# B&R Automation Studio project ControlObjectModeling
Automation Studio 4.2.10.53 SP

## Configuration Config1

CPU 4PP065.0351-P74, AutomationRuntime D4.26, Build 4.1.2, Vc V4.26.5, Safety 0.0

### Task classes (Cpu.sw)
```
Cyclic#2 (cycle 20000 us, tolerance 20000 us):
  Program <- Program.prg
Binaries: TCData, iomap, Role, sysconf, arconfig, asfw, User, ashwd
Libraries: MotorContr
```

### Hardware
```
4PP065_0351_P74 : 4PP065.0351-P74 v1.0.3.0
  Connector IF4:
    EplInterfaceRedundant = 0
    EplEthInterfaceRedundant = 0
  Connector IF5:
    ActivateDevice = 1
  ConfigurationID = Lab1_Config1
  Simulation = 1
  Cyclic1Duration = 10000
  Cyclic1Tolerance = 10000
  Cyclic2Duration = 20000
  Cyclic2Tolerance = 20000
  Cyclic3Duration = 50000
  Cyclic3Tolerance = 50000
  Cyclic4Duration = 100000
  Cyclic4Tolerance = 100000
  Cyclic5Duration = 200000
  Cyclic5Tolerance = 200000
  Cyclic6Duration = 500000
  Cyclic6Tolerance = 500000
  Cyclic7Duration = 1000000
  Cyclic7Tolerance = 1000000
  Cyclic8Duration = 10000
  Cyclic8Tolerance = 30000000
```

## Logical view

Binary libraries used (declarations not repeated): operator, runtime, astime, AsIecCon

### Package Logical/Libraries - Global libraries

### Library Logical/Libraries/MotorContr (ANSIC)

#### MotorContr.fun - Exported functions and function blocks
```iecst
FUNCTION_BLOCK FB_Regulator (*Regulator functional block*) (*$GROUP=User,$CAT=User,$GROUPICON=User.png,$CATICON=User.png*)
	VAR_INPUT
		e : REAL; (*Mismatch between the reference action and the real speed of rotation of the DCM shaft [rpm]*)
	END_VAR
	VAR_OUTPUT
		u : REAL; (*Voltage supplied to the DCM input [V]*)
	END_VAR
	VAR
		k_p : REAL; (*Regulator proportional gain*)
		k_i : REAL; (*Integral gain of the regulator*)
		integrator : FB_Integrator; (*Integrator*)
		iyOld : REAL; (*Storing the previous value of the anti-accumulation scheme*)
		max_abs_value : REAL; (*Limit block boundary [B]*)
		dt : REAL; (*Calculation step [s]*)
		e_p : REAL; (*Temporary variable [rpm]*)
	END_VAR
END_FUNCTION_BLOCK

FUNCTION_BLOCK FB_Motor (*Motor functional block*) (*$GROUP=User,$CAT=User,$GROUPICON=User.png,$CATICON=User.png*)
	VAR_INPUT
		u : REAL; (*Input voltage [V]*)
	END_VAR
	VAR_OUTPUT
		w : REAL; (*Rotation frequency [rpm]*)
		phi : REAL; (*Position [rad]*)
	END_VAR
	VAR
		integrator : FB_Integrator; (*Integrator*)
		Tm : REAL; (*Electromechanical time constant [s]*)
		ke : REAL; (*Constant EMF of the motor [V * min/rev]*)
		dt : REAL; (*Calculation step [s]*)
	END_VAR
END_FUNCTION_BLOCK

FUNCTION_BLOCK FB_Integrator (*Integrator functional block*) (*$GROUP=User,$CAT=User,$GROUPICON=User.png,$CATICON=User.png*)
	VAR_INPUT
		in : REAL; (*Integrator input*)
	END_VAR
	VAR_OUTPUT
		out : REAL; (*Integrator output*)
	END_VAR
	VAR
		dt : REAL; (*Calculation step [s]*)
	END_VAR
END_FUNCTION_BLOCK
```

### Program Logical/Program (ANSIC)

#### Variables.var
```iecst
VAR
	fb_motor_1 : FB_Motor; (*DCM model*)
	fb_motor_2 : FB_Motor; (*DCM model*)
	fb_regulator : FB_Regulator; (*Regulator model*)
	enable : BOOL; (*Integral gain of the regulator*)
	counter : REAL; (*Counter*)
	speed : REAL; (*Speed setpoint*)
END_VAR
```

#### Main.c
```c
#include <bur/plctypes.h>

#ifdef _DEFAULT_INCLUDES
	#include <AsDefault.h>
#endif

void _INIT ProgramInit(void)
{
	enable = 1;
	counter = 0;
	speed = 0;

	fb_regulator.dt = 0.02;
	fb_regulator.k_i = 16;
	fb_regulator.k_p = 0.64;
	fb_regulator.max_abs_value = 24;

	fb_motor_1.dt = 0.02;
	fb_motor_1.ke = 16;
	fb_motor_1.Tm = 0.04;

	fb_motor_2.dt = 0.02;
	fb_motor_2.ke = 16;
	fb_motor_2.Tm = 0.04;
}

void _CYCLIC ProgramCyclic(void)
{
	if(enable == 1)
	{
		counter += 10;
		if(counter >= 10000 && counter <= 15000) speed = 5;
		else speed = 0;
	}
	else speed = 0;

	fb_regulator.e = speed - fb_motor_1.w;
	FB_Regulator(&(fb_regulator));

	fb_motor_1.u = fb_regulator.u*fb_motor_1.ke;
	fb_motor_2.u = speed*fb_motor_2.ke;
	FB_Motor(&(fb_motor_1));
	FB_Motor(&(fb_motor_2));
}

void _EXIT ProgramExit(void)
{
	// Insert code here

}
```

Listed in the project but not available here: Logical/Global.typ, Logical/Global.var, Logical/Libraries/MotorContr/Types.typ, Logical/Libraries/MotorContr/Constants.var, Logical/Libraries/MotorContr/FB_Motor.c, Logical/Libraries/MotorContr/FB_Regulator.c, Logical/Libraries/MotorContr/FB_Integrator.c
